// TIA Portal V20 export
TYPE "LKinCtrl_typeHMIInterface"
// stored: Access Published
   STRUCT
      teachKinematics : "LKinCtrl_TeachKinematics_typeHMIInterface";
      editors : "LKinCtrl_Editor_typeHMIInterface";
      diagnostics : "LKinCtrl_Diagnostics_typeHMIInterface";
   END_STRUCT;
END_TYPE
